// TwinCAT 3 PLC project SerialCom
// ProgramVersion: 3.1.4023.0
// libraries:
//   Tc2_SerialCom, * (Beckhoff Automation GmbH)
//   Tc2_Standard, * (Beckhoff Automation GmbH)
//   Tc2_System, * (Beckhoff Automation GmbH)
//   Tc3_Module, * (Beckhoff Automation GmbH)
// project tree:
//   / CommTask.TcTTO, PlcTask.TcTTO
//   GVLs/ SerialComm.TcGVL
//   POUs/ BackgroungCommProgram.TcPOU, MAIN.TcPOU
//   POUs/FB%27s/ SerialCom.TcPOU (not stored)

CONFIGURATION SerialCom
    RESOURCE PLC ON TwinCAT3
        TASK CommTask(INTERVAL := T#2ms, PRIORITY := 19);
        TASK PlcTask(INTERVAL := T#10ms, PRIORITY := 20);
        PROGRAM BackgroungCommProgram WITH CommTask : BackgroungCommProgram;
        PROGRAM MAIN WITH PlcTask : MAIN;
    END_RESOURCE
END_CONFIGURATION

// ---- GVLs/SerialComm.TcGVL
{attribute 'qualified_only'}
VAR_GLOBAL
(* Buffer Variable *)
RxBufferPcCom		: ComBuffer;	(* Receive data buffer; used with all receive function blocks *)
TxBufferPcCom		: ComBuffer;	(* Transmit data buffer; used with all receive function blocks *)
END_VAR

// ---- POUs/BackgroungCommProgram.TcPOU
PROGRAM BackgroungCommProgram
VAR
(* Comm I/O Variable *)
(* I/O variables for a PC-COM port *)
stIn_PcCom AT %I* : PcComInData; (* linked to the port in the TwinCAT System Manager *)
stOut_PcCom AT %Q* : PcComOutData; (* linked to the port in the TwinCAT System Manager *)
	
(* Background communication with the PC COM port device *)
fbPcComCtrl			: SerialLineControl;
bPcComCtrlError		: BOOL;
ePcComCtrlErrorID	: ComError_t;	


END_VAR

(*
The SerialLineControl function block is supposed to be called in every PLC cycle.
It communicates with the serial line hardware device and transmits or receives data 
*)

fbPcComCtrl(
	Mode:= SERIALLINEMODE_PC_COM_PORT, 
	pComIn:= ADR(stIn_PcCom), 
	pComOut:= ADR(stOut_PcCom), 
	SizeComIn:= UINT_TO_INT(SIZEOF(stIn_PcCom)), 
	Error=> , 
	ErrorID=> , 
	TxBuffer:= SerialComm.TxBufferPcCom, 
	RxBuffer:= SerialComm.RxBufferPcCom);
	
IF fbPcComCtrl.Error THEN
	bPcComCtrlError := TRUE;
	ePcComCtrlErrorID := fbPcComCtrl.ErrorID;
END_IF

END_PROGRAM

// ---- POUs/MAIN.TcPOU
PROGRAM MAIN
VAR
	fbSerialCommInstance1 : SerialCom;
	sRecieveString : STRING;
	bRecieveError : BOOL;
	bSendBusy: BOOL;
	eSendError: INT;
	sSendData : STRING;
	bsendTrigger: BOOL;
	STxBuffer: INT;
	tSendTime: INT;
	sizeoff : UINT;
	bRecieveReset: BOOL;
END_VAR

(* Send & Recieve String Data *)
fbSerialCommInstance1(bSendData:= bsendTrigger,
					  bReset := bRecieveReset,
					  TxBuffer := SerialComm.TxBufferPcCom,
					  sSendPrefix:='$01',
					  sSendSuffix:='$02',
					  sSendString:=sSendData,
					  bSendBusy =>bSendBusy,
					  eSendError =>eSendError,
					  RxBuffer := SerialComm.RxBufferPcCom,
					  sReceiveString =>sRecieveString,
					  sReceivePrefix:='$01',
					  sReceiveSuffix:='$02',
					  tReceiveTimeOut := T#1S,
					  bReset :=bRecieveError,
					  bReceiveStringData =>,
					  bReceiveBusy =>,
					  eReceiveError =>,
					  bReceiveTimeOut =>
					  );

END_PROGRAM
